FUNCTION_BLOCK FB_AbstractChild EXTENDS FB_Abstract
VAR_INPUT
END_VAR
VAR_OUTPUT
END_VAR
VAR
END_VAR

{warning 'Add method implementation '} //  Auto generated due to child class being Abstract
METHOD PROTECTED M_Init : BOOL
END_METHOD

END_FUNCTION_BLOCK

(* stored: Version 1.1.0.1
   POU FB_AbstractChild: Id {fca5e974-7120-4707-865c-037c45120a8f}, SpecialFunc None
   Method M_Init: Id {ef0cb9a8-dc0b-43c8-929e-629171d6e113} *)
